INTERFACE I_StructureMembers

METHOD PUBLIC Accept
VAR_INPUT
	Visitor : I_DatatypeVisitor;
END_VAR
END_METHOD

METHOD PUBLIC GetMemberEnumerator : I_KeyValueForwardEnumerator
VAR_INPUT
END_VAR
END_METHOD

METHOD PUBLIC TryGetMemberByName : BOOL
VAR_INPUT
	Name : T_MAXSTRING;
	Destination : REFERENCE TO I_Datatype;
END_VAR
END_METHOD

END_INTERFACE

(* stored: Version 1.1.0.1, ProductVersion 3.1.4024.12
   Itf I_StructureMembers: Id {725904a6-8cf8-48b8-a6ca-3bfc37513b86}
   Method Accept: Id {9fbe2c54-4e72-4a46-9ac6-f053d2bfd090}
   Method GetMemberEnumerator: Id {c78504c1-5fa4-4ffc-9d04-5cb07e1c5e21}
   Method TryGetMemberByName: Id {acaf4a37-304c-475a-a555-d6589588d23e} *)
